(* IEC 61131-3 sources: Lasal/CPU_5344_V01/Class/OperationLineV2, 1 file *)

(* ---- OperationLineV2.st ---- *)
(*!
<Class
	Name               = "OperationLineV2"
	Revision           = "0.0"
	RealtimeTask       = "false"
	CyclicTask         = "false"
	BackgroundTask     = "false"
	Sigmatek           = "false"
	OSInterface        = "false"
	HighPriority       = "false"
	Automatic          = "false"
	UpdateMode         = "Prescan"
	SharedCommandTable = "true"
	Objectsize         = "(390,360)">
	<Channels>
		<Server Name="amount" Visualized="true" Initialize="false" WriteProtected="false" Retentive="false"/>
		<Server Name="ClassSvr" Visualized="false" Initialize="false" WriteProtected="true" Retentive="false"/>
		<Server Name="operationId" Visualized="true" Initialize="false" WriteProtected="false" Retentive="false"/>
		<Server Name="operationType" Visualized="true" Initialize="false" WriteProtected="false" Retentive="false"/>
		<Server Name="pitch" Visualized="true" Initialize="false" WriteProtected="false" Retentive="false"/>
		<Server Name="rnr" Visualized="true" Initialize="false" WriteProtected="false" Retentive="false"/>
		<Server Name="xPos" Visualized="true" Initialize="false" WriteProtected="false" Retentive="false"/>
		<Server Name="yPos" Visualized="true" Initialize="false" WriteProtected="false" Retentive="false"/>
		<Server Name="zPos" Visualized="true" Initialize="false" WriteProtected="false" Retentive="false"/>
	</Channels>
</Class>
*)
OperationLineV2 : CLASS
  //Servers:
	ClassSvr 	: SvrChCmd_DINT;
	rnr 	: SvrCh_DINT;
	xPos 	: SvrCh_DINT;
	yPos 	: SvrCh_DINT;
	zPos 	: SvrCh_DINT;
	amount 	: SvrCh_DINT;
	pitch 	: SvrCh_DINT;
	operationType 	: SvrCh_DINT;
	operationId 	: SvrCh_DINT;
  //Clients:
  //Variables:
		ptr 	: ^ProductsDbV2::tRecipeLine;
		ptrHeigth 	: ^DINT;
		useHeigth 	: DINT;
  //Functions:

	FUNCTION GLOBAL WritePtr
		VAR_INPUT
			iPtr 	: ^ProductsDbV2::tRecipeLine;
			iPtrProdHeigth 	: ^DINT;
			iUseHeigth 	: DINT;
		END_VAR;

	FUNCTION WriteServers;

	FUNCTION VIRTUAL GLOBAL xPos::Write
		VAR_INPUT
			input (EAX) 	: DINT;
		END_VAR
		VAR_OUTPUT
			result (EAX) 	: DINT;
		END_VAR;

	FUNCTION VIRTUAL GLOBAL yPos::Write
		VAR_INPUT
			input (EAX) 	: DINT;
		END_VAR
		VAR_OUTPUT
			result (EAX) 	: DINT;
		END_VAR;

	FUNCTION VIRTUAL GLOBAL zPos::Write
		VAR_INPUT
			input (EAX) 	: DINT;
		END_VAR
		VAR_OUTPUT
			result (EAX) 	: DINT;
		END_VAR;

	FUNCTION VIRTUAL GLOBAL amount::Write
		VAR_INPUT
			input (EAX) 	: DINT;
		END_VAR
		VAR_OUTPUT
			result (EAX) 	: DINT;
		END_VAR;

	FUNCTION VIRTUAL GLOBAL pitch::Write
		VAR_INPUT
			input (EAX) 	: DINT;
		END_VAR
		VAR_OUTPUT
			result (EAX) 	: DINT;
		END_VAR;

	FUNCTION VIRTUAL GLOBAL operationType::Write
		VAR_INPUT
			input (EAX) 	: DINT;
		END_VAR
		VAR_OUTPUT
			result (EAX) 	: DINT;
		END_VAR;

	FUNCTION VIRTUAL GLOBAL operationId::Write
		VAR_INPUT
			input (EAX) 	: DINT;
		END_VAR
		VAR_OUTPUT
			result (EAX) 	: DINT;
		END_VAR;
  //Tables:
	FUNCTION @STD
		VAR_OUTPUT
			ret_code	: CONFSTATES;
		END_VAR;
	FUNCTION GLOBAL TAB @CT_;
END_CLASS;

FUNCTION VIRTUAL GLOBAL OperationLineV2::xPos::Write
	VAR_INPUT
		input (EAX) 	: DINT;
	END_VAR
	VAR_OUTPUT
		result (EAX) 	: DINT;
	END_VAR

  if ptr <> NIL then
    xPos := input;
    ptr^.xpos := xPos;
    IF useHeigth= 1 THEN //method to always write y pos to half width
      zPos.Write(input:=ptrHeigth^/2);
    END_IF;
    result := xPos;
  else
    result := ACCESS_DENIED;
  end_if;

END_FUNCTION

FUNCTION VIRTUAL GLOBAL OperationLineV2::yPos::Write
	VAR_INPUT
		input (EAX) 	: DINT;
	END_VAR
	VAR_OUTPUT
		result (EAX) 	: DINT;
	END_VAR

  if ptr <> NIL then
    yPos := input;
    ptr^.ypos := yPos;
    result := yPos;
  else
    result := ACCESS_DENIED;
  end_if;

END_FUNCTION

FUNCTION VIRTUAL GLOBAL OperationLineV2::zPos::Write
	VAR_INPUT
		input (EAX) 	: DINT;
	END_VAR
	VAR_OUTPUT
		result (EAX) 	: DINT;
	END_VAR

  if ptr <> NIL then
    zPos := input;
    ptr^.zpos := zPos;
    result := zPos;
  else
    result := ACCESS_DENIED;
  end_if;

END_FUNCTION

FUNCTION VIRTUAL GLOBAL OperationLineV2::operationType::Write
	VAR_INPUT
		input (EAX) 	: DINT;
	END_VAR
	VAR_OUTPUT
		result (EAX) 	: DINT;
	END_VAR

  if ptr <> NIL then
    operationType := input;
    ptr^.operations := operationType$::tBewerkingType;
    IF useHeigth= 1 THEN //method to always write y pos to half width
      zPos.Write(input:=ptrHeigth^/2);
    END_IF;
    result := operationType;
  else
    result := ACCESS_DENIED;
  end_if;

END_FUNCTION

FUNCTION GLOBAL OperationLineV2::WritePtr
	VAR_INPUT
		iPtr 	: ^ProductsDbV2::tRecipeLine;
		iPtrProdHeigth 	: ^DINT;
		iUseHeigth 	: DINT;
	END_VAR

  ptr := iPtr;
  ptrHeigth := iPtrProdHeigth;
  useHeigth := iUseHeigth;

  WriteServers();

END_FUNCTION

FUNCTION OperationLineV2::WriteServers

  if ptr <> NIL then
    xPos := ptr^.xpos;
    yPos := ptr^.ypos;
    zPos := ptr^.zpos;
    operationId := ptr^.operationId;
    amount := ptr^.amount;
    pitch := ptr^.pitch;
    operationType := ptr^.operations$DINT;
  end_if;

END_FUNCTION

FUNCTION VIRTUAL GLOBAL OperationLineV2::amount::Write
	VAR_INPUT
		input (EAX) 	: DINT;
	END_VAR
	VAR_OUTPUT
		result (EAX) 	: DINT;
	END_VAR

  if ptr <> NIL then
	  amount := input;
    ptr^.amount := amount;
	  result := amount;
  else
    result := ACCESS_DENIED;
  end_if;

END_FUNCTION

FUNCTION VIRTUAL GLOBAL OperationLineV2::pitch::Write
	VAR_INPUT
		input (EAX) 	: DINT;
	END_VAR
	VAR_OUTPUT
		result (EAX) 	: DINT;
	END_VAR

  if ptr <> NIL then
	  pitch := input;
    ptr^.pitch := pitch;
	  result := pitch;
  else
    result := ACCESS_DENIED;
  end_if;

END_FUNCTION

FUNCTION VIRTUAL GLOBAL OperationLineV2::operationId::Write
	VAR_INPUT
		input (EAX) 	: DINT;
	END_VAR
	VAR_OUTPUT
		result (EAX) 	: DINT;
	END_VAR

  if ptr <> NIL then
    operationId := input;
    ptr^.operationId := operationId;
    result := operationId;
  else
    result := ACCESS_DENIED;
  end_if;

END_FUNCTION
